SYSTEM test
  (* Version 1.0, 2022-11-09, franz *)
  APPLICATION testApp
  END_APPLICATION
  APPLICATION mapping_DataPanel
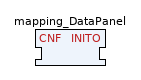
    SUBAPPLICATION mapping_DataPanel (* mapping_DataPanel *)
      EVENT_INPUT
        CNF;
      END_EVENT
      EVENT_OUTPUT
        INITO;
      END_EVENT
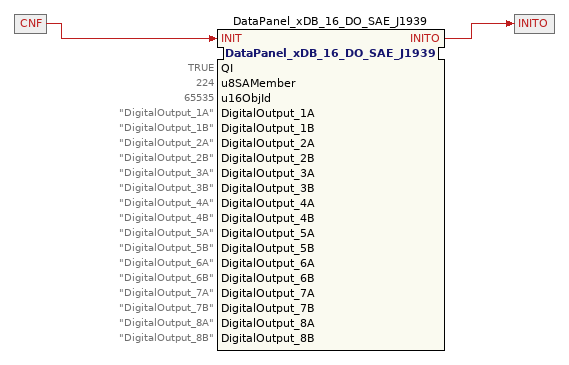
      FBS
        DataPanel_xDB_16_DO_SAE_J1939 : DataPanel_xDB_16_DO_SAE_J1939(QI := TRUE, u8SAMember := 224, u16ObjId := 65535, DigitalOutput_1A := "DigitalOutput_1A", DigitalOutput_1B := "DigitalOutput_1B", DigitalOutput_2A := "DigitalOutput_2A", DigitalOutput_2B := "DigitalOutput_2B", DigitalOutput_3A := "DigitalOutput_3A", DigitalOutput_3B := "DigitalOutput_3B", DigitalOutput_4A := "DigitalOutput_4A", DigitalOutput_4B := "DigitalOutput_4B", DigitalOutput_5A := "DigitalOutput_5A", DigitalOutput_5B := "DigitalOutput_5B", DigitalOutput_6A := "DigitalOutput_6A", DigitalOutput_6B := "DigitalOutput_6B", DigitalOutput_7A := "DigitalOutput_7A", DigitalOutput_7B := "DigitalOutput_7B", DigitalOutput_8A := "DigitalOutput_8A", DigitalOutput_8B := "DigitalOutput_8B");
      END_FBS
      EVENT_CONNECTIONS
        CNF TO DataPanel_xDB_16_DO_SAE_J1939.INIT;
        DataPanel_xDB_16_DO_SAE_J1939.INITO TO INITO;
      END_CONNECTIONS
    END_SUBAPPLICATION
  END_APPLICATION
  APPLICATION mapping_Softkeys
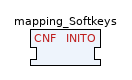
    SUBAPPLICATION mapping_Softkeys (* mapping_Softkeys *)
      EVENT_INPUT
        CNF;
      END_EVENT
      EVENT_OUTPUT
        INITO;
      END_EVENT
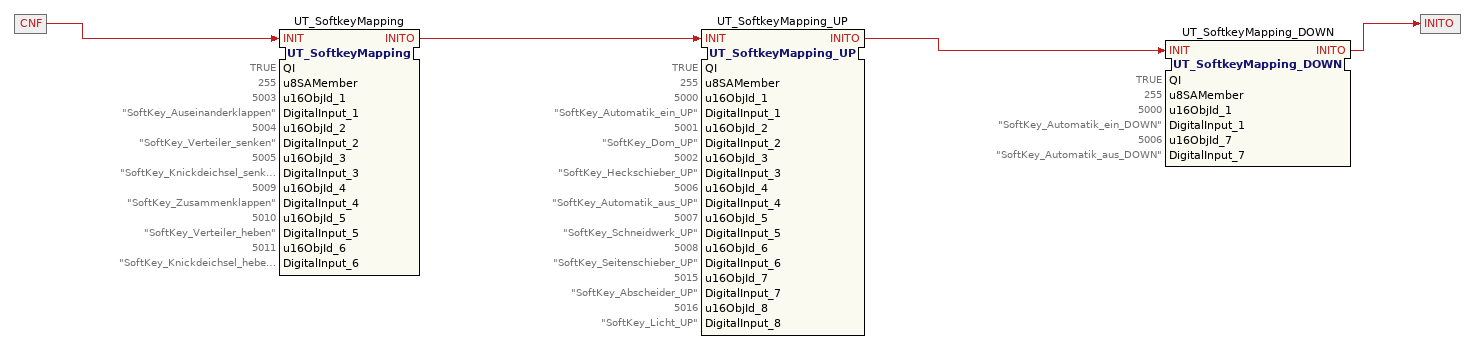
      FBS
        UT_SoftkeyMapping_DOWN : UT_SoftkeyMapping_DOWN(QI := TRUE, u8SAMember := 255, u16ObjId_1 := 5000, DigitalInput_1 := "SoftKey_Automatik_ein_DOWN", u16ObjId_7 := 5006, DigitalInput_7 := "SoftKey_Automatik_aus_DOWN");
        UT_SoftkeyMapping_UP : UT_SoftkeyMapping_UP(QI := TRUE, u8SAMember := 255, u16ObjId_1 := 5000, DigitalInput_1 := "SoftKey_Automatik_ein_UP", u16ObjId_2 := 5001, DigitalInput_2 := "SoftKey_Dom_UP", u16ObjId_3 := 5002, DigitalInput_3 := "SoftKey_Heckschieber_UP", u16ObjId_4 := 5006, DigitalInput_4 := "SoftKey_Automatik_aus_UP", u16ObjId_5 := 5007, DigitalInput_5 := "SoftKey_Schneidwerk_UP", u16ObjId_6 := 5008, DigitalInput_6 := "SoftKey_Seitenschieber_UP", u16ObjId_7 := 5015, DigitalInput_7 := "SoftKey_Abscheider_UP", u16ObjId_8 := 5016, DigitalInput_8 := "SoftKey_Licht_UP");
        UT_SoftkeyMapping : UT_SoftkeyMapping(QI := TRUE, u8SAMember := 255, u16ObjId_1 := 5003, DigitalInput_1 := "SoftKey_Auseinanderklappen", u16ObjId_2 := 5004, DigitalInput_2 := "SoftKey_Verteiler_senken", u16ObjId_3 := 5005, DigitalInput_3 := "SoftKey_Knickdeichsel_senken", u16ObjId_4 := 5009, DigitalInput_4 := "SoftKey_Zusammenklappen", u16ObjId_5 := 5010, DigitalInput_5 := "SoftKey_Verteiler_heben", u16ObjId_6 := 5011, DigitalInput_6 := "SoftKey_Knickdeichsel_heben");
      END_FBS
      EVENT_CONNECTIONS
        UT_SoftkeyMapping_UP.INITO TO UT_SoftkeyMapping_DOWN.INIT;
        UT_SoftkeyMapping.INITO TO UT_SoftkeyMapping_UP.INIT;
        UT_SoftkeyMapping_DOWN.INITO TO INITO;
        CNF TO UT_SoftkeyMapping.INIT;
      END_CONNECTIONS
    END_SUBAPPLICATION
  END_APPLICATION
  APPLICATION Klappen
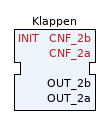
    SUBAPPLICATION Klappen (* Klappen *)
      EVENT_INPUT
        INIT;
      END_EVENT
      EVENT_OUTPUT
        CNF_2b;
        CNF_2a;
      END_EVENT
      VAR_OUTPUT
        OUT_2b : BOOL;
        OUT_2a : BOOL;
      END_VAR
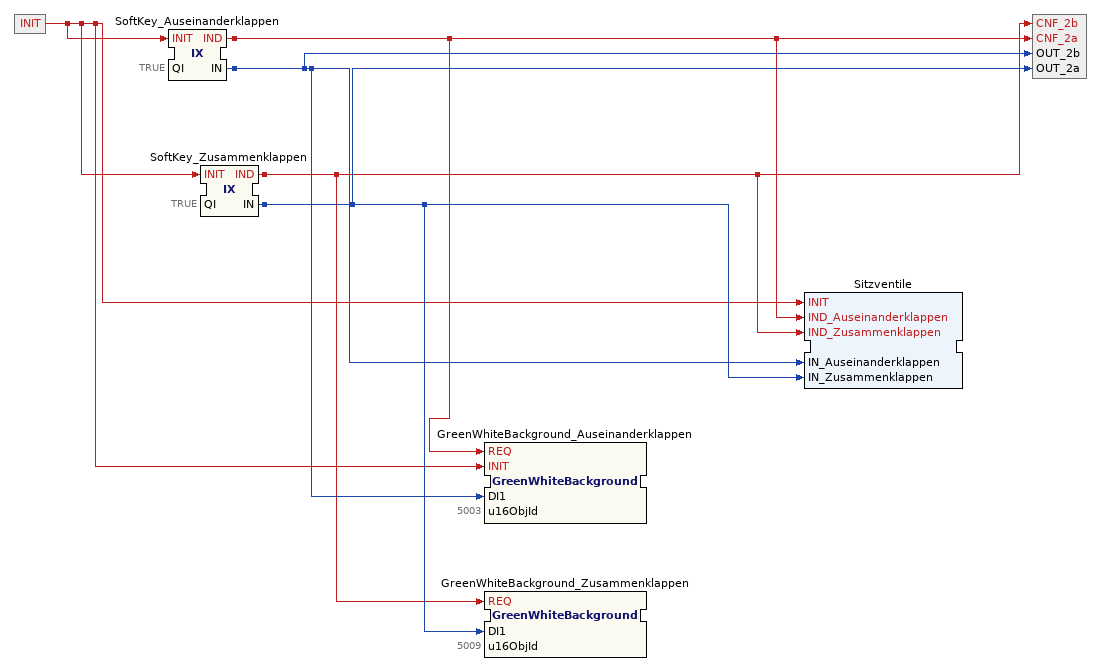
      FBS
        SoftKey_Auseinanderklappen : IX(QI := TRUE);
        GreenWhiteBackground_Auseinanderklappen : GreenWhiteBackground(u16ObjId := 5003);
        SoftKey_Zusammenklappen : IX(QI := TRUE);
        GreenWhiteBackground_Zusammenklappen : GreenWhiteBackground(u16ObjId := 5009);
      END_FBS
      SUBAPPLICATION Sitzventile (* Sitzventile *)
        EVENT_INPUT
          INIT;
          IND_Auseinanderklappen;
          IND_Zusammenklappen;
        END_EVENT
        VAR_INPUT
          IN_Auseinanderklappen : BOOL;
          IN_Zusammenklappen : BOOL;
        END_VAR
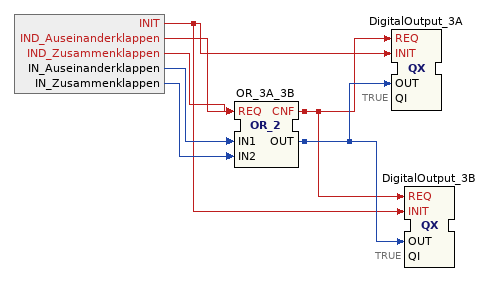
        FBS
          DigitalOutput_3B : QX(QI := TRUE);
          DigitalOutput_3A : QX(QI := TRUE);
          OR_3A_3B : OR_2; {SET_ATTRIBUTE(PinComment, IN1:Auseinanderklappen)} {SET_ATTRIBUTE(PinComment, IN2:Zusammenklappen)}
        END_FBS
        EVENT_CONNECTIONS
          OR_3A_3B.CNF TO DigitalOutput_3B.REQ;
          OR_3A_3B.CNF TO DigitalOutput_3A.REQ;
          INIT TO DigitalOutput_3B.INIT;
          INIT TO DigitalOutput_3A.INIT;
          IND_Auseinanderklappen TO OR_3A_3B.REQ;
          IND_Zusammenklappen TO OR_3A_3B.REQ;
        END_CONNECTIONS
        DATA_CONNECTIONS
          OR_3A_3B.OUT TO DigitalOutput_3B.OUT;
          OR_3A_3B.OUT TO DigitalOutput_3A.OUT;
          IN_Auseinanderklappen TO OR_3A_3B.IN1;
          IN_Zusammenklappen TO OR_3A_3B.IN2;
        END_CONNECTIONS
      END_SUBAPPLICATION
      EVENT_CONNECTIONS
        SoftKey_Auseinanderklappen.IND TO GreenWhiteBackground_Auseinanderklappen.REQ;
        INIT TO SoftKey_Auseinanderklappen.INIT;
        SoftKey_Auseinanderklappen.IND TO CNF_2b;
        INIT TO SoftKey_Zusammenklappen.INIT;
        SoftKey_Zusammenklappen.IND TO CNF_2a;
        INIT TO GreenWhiteBackground_Auseinanderklappen.INIT;
        INIT TO Sitzventile.INIT;
        SoftKey_Auseinanderklappen.IND TO Sitzventile.IND_Auseinanderklappen;
        SoftKey_Zusammenklappen.IND TO Sitzventile.IND_Zusammenklappen;
        SoftKey_Zusammenklappen.IND TO GreenWhiteBackground_Zusammenklappen.REQ;
      END_CONNECTIONS
      DATA_CONNECTIONS
        SoftKey_Auseinanderklappen.IN TO GreenWhiteBackground_Auseinanderklappen.DI1;
        SoftKey_Auseinanderklappen.IN TO OUT_2b;
        SoftKey_Zusammenklappen.IN TO OUT_2a;
        SoftKey_Auseinanderklappen.IN TO Sitzventile.IN_Auseinanderklappen;
        SoftKey_Zusammenklappen.IN TO Sitzventile.IN_Zusammenklappen;
        SoftKey_Zusammenklappen.IN TO GreenWhiteBackground_Zusammenklappen.DI1;
      END_CONNECTIONS
    END_SUBAPPLICATION
  END_APPLICATION
  APPLICATION Vorsteuerventil_2A
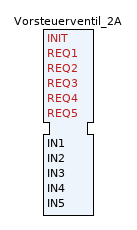
    SUBAPPLICATION Vorsteuerventil_2A (* Vorsteuerventil_2A *)
      EVENT_INPUT
        INIT;
        REQ1;
        REQ2;
        REQ3;
        REQ4;
        REQ5;
      END_EVENT
      VAR_INPUT
        IN1 : BOOL;
        IN2 : BOOL;
        IN3 : BOOL;
        IN4 : BOOL;
        IN5 : BOOL;
      END_VAR
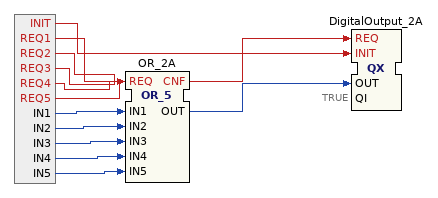
      FBS
        DigitalOutput_2A : QX(QI := TRUE);
        OR_2A : OR_5;
      END_FBS
      EVENT_CONNECTIONS
        OR_2A.CNF TO DigitalOutput_2A.REQ;
        INIT TO DigitalOutput_2A.INIT;
        REQ1 TO OR_2A.REQ;
        REQ2 TO OR_2A.REQ;
        REQ3 TO OR_2A.REQ;
        REQ4 TO OR_2A.REQ;
        REQ5 TO OR_2A.REQ;
      END_CONNECTIONS
      DATA_CONNECTIONS
        OR_2A.OUT TO DigitalOutput_2A.OUT;
        IN1 TO OR_2A.IN1;
        IN2 TO OR_2A.IN2;
        IN3 TO OR_2A.IN3;
        IN4 TO OR_2A.IN4;
        IN5 TO OR_2A.IN5;
      END_CONNECTIONS
    END_SUBAPPLICATION
  END_APPLICATION
  APPLICATION Verteiler
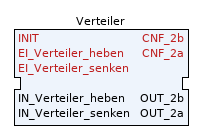
    SUBAPPLICATION Verteiler (* Verteiler *)
      EVENT_INPUT
        INIT;
        EI_Verteiler_heben;
        EI_Verteiler_senken;
      END_EVENT
      EVENT_OUTPUT
        CNF_2b;
        CNF_2a;
      END_EVENT
      VAR_INPUT
        IN_Verteiler_heben : BOOL;
        IN_Verteiler_senken : BOOL;
      END_VAR
      VAR_OUTPUT
        OUT_2b : BOOL;
        OUT_2a : BOOL;
      END_VAR
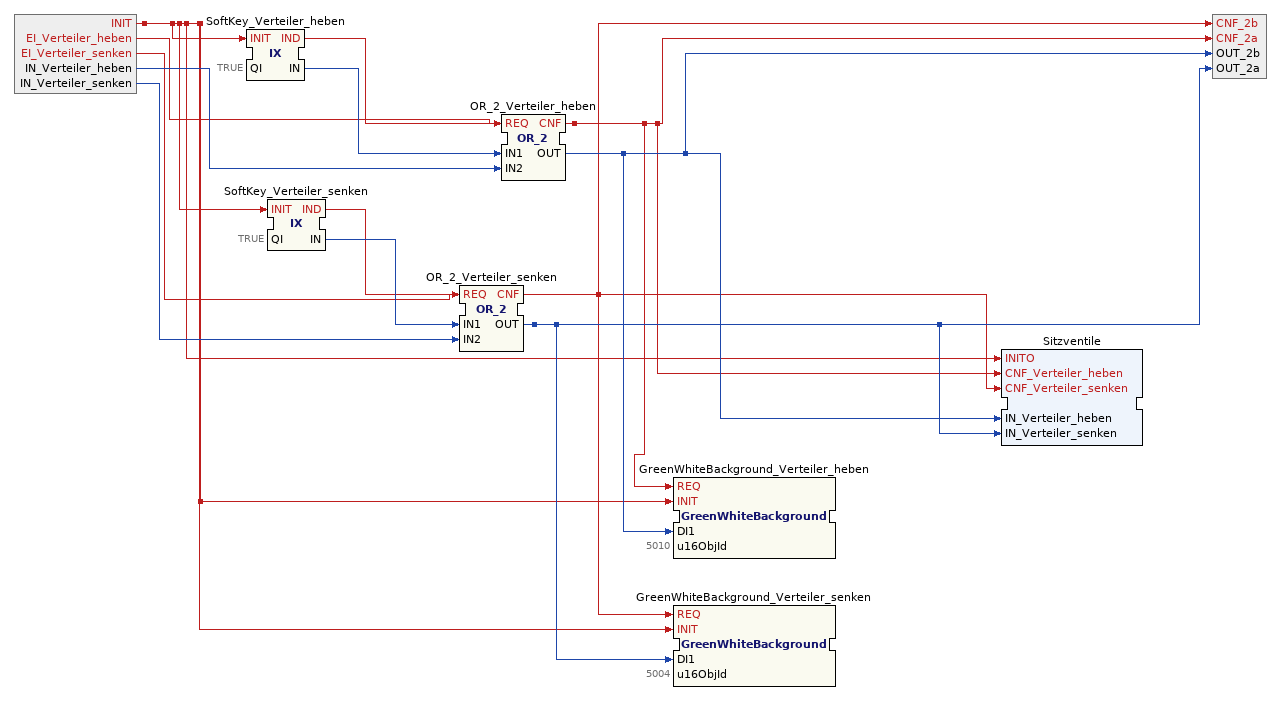
      FBS
        OR_2_Verteiler_senken : OR_2;
        SoftKey_Verteiler_heben : IX(QI := TRUE);
        OR_2_Verteiler_heben : OR_2;
        GreenWhiteBackground_Verteiler_heben : GreenWhiteBackground(u16ObjId := 5010);
        SoftKey_Verteiler_senken : IX(QI := TRUE);
        GreenWhiteBackground_Verteiler_senken : GreenWhiteBackground(u16ObjId := 5004);
      END_FBS
      SUBAPPLICATION Sitzventile (* Sitzventile *)
        EVENT_INPUT
          INITO;
          CNF_Verteiler_heben;
          CNF_Verteiler_senken;
        END_EVENT
        VAR_INPUT
          IN_Verteiler_heben : BOOL;
          IN_Verteiler_senken : BOOL;
        END_VAR
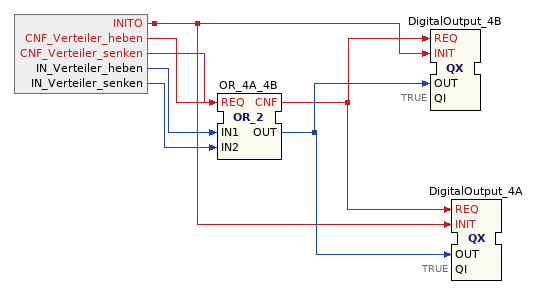
        FBS
          OR_4A_4B : OR_2; {SET_ATTRIBUTE(PinComment, IN1:Verteiler_heben)} {SET_ATTRIBUTE(PinComment, IN2:Verteiler_senken)}
          DigitalOutput_4B : QX(QI := TRUE);
          DigitalOutput_4A : QX(QI := TRUE);
        END_FBS
        EVENT_CONNECTIONS
          OR_4A_4B.CNF TO DigitalOutput_4B.REQ;
          OR_4A_4B.CNF TO DigitalOutput_4A.REQ;
          CNF_Verteiler_heben TO OR_4A_4B.REQ;
          CNF_Verteiler_senken TO OR_4A_4B.REQ;
          INITO TO DigitalOutput_4B.INIT;
          INITO TO DigitalOutput_4A.INIT;
        END_CONNECTIONS
        DATA_CONNECTIONS
          OR_4A_4B.OUT TO DigitalOutput_4B.OUT;
          OR_4A_4B.OUT TO DigitalOutput_4A.OUT;
          IN_Verteiler_heben TO OR_4A_4B.IN1;
          IN_Verteiler_senken TO OR_4A_4B.IN2;
        END_CONNECTIONS
      END_SUBAPPLICATION
      EVENT_CONNECTIONS
        SoftKey_Verteiler_senken.IND TO OR_2_Verteiler_senken.REQ;
        SoftKey_Verteiler_heben.IND TO OR_2_Verteiler_heben.REQ;
        OR_2_Verteiler_heben.CNF TO GreenWhiteBackground_Verteiler_heben.REQ;
        INIT TO SoftKey_Verteiler_heben.INIT;
        INIT TO SoftKey_Verteiler_senken.INIT;
        INIT TO Sitzventile.INITO;
        OR_2_Verteiler_senken.CNF TO GreenWhiteBackground_Verteiler_senken.REQ;
        INIT TO GreenWhiteBackground_Verteiler_heben.INIT;
        INIT TO GreenWhiteBackground_Verteiler_senken.INIT;
        OR_2_Verteiler_heben.CNF TO CNF_2a;
        OR_2_Verteiler_senken.CNF TO CNF_2b;
        OR_2_Verteiler_heben.CNF TO Sitzventile.CNF_Verteiler_heben;
        OR_2_Verteiler_senken.CNF TO Sitzventile.CNF_Verteiler_senken;
        EI_Verteiler_heben TO OR_2_Verteiler_heben.REQ;
        EI_Verteiler_senken TO OR_2_Verteiler_senken.REQ;
      END_CONNECTIONS
      DATA_CONNECTIONS
        SoftKey_Verteiler_senken.IN TO OR_2_Verteiler_senken.IN1;
        SoftKey_Verteiler_heben.IN TO OR_2_Verteiler_heben.IN1;
        OR_2_Verteiler_heben.OUT TO GreenWhiteBackground_Verteiler_heben.DI1;
        IN_Verteiler_senken TO OR_2_Verteiler_senken.IN2;
        IN_Verteiler_heben TO OR_2_Verteiler_heben.IN2;
        OR_2_Verteiler_heben.OUT TO Sitzventile.IN_Verteiler_heben;
        OR_2_Verteiler_senken.OUT TO Sitzventile.IN_Verteiler_senken;
        OR_2_Verteiler_senken.OUT TO GreenWhiteBackground_Verteiler_senken.DI1;
        OR_2_Verteiler_heben.OUT TO OUT_2b;
        OR_2_Verteiler_senken.OUT TO OUT_2a;
      END_CONNECTIONS
    END_SUBAPPLICATION
  END_APPLICATION
  APPLICATION Knickdeichsel
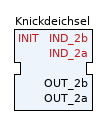
    SUBAPPLICATION Knickdeichsel (* Knickdeichsel *)
      EVENT_INPUT
        INIT;
      END_EVENT
      EVENT_OUTPUT
        IND_2b;
        IND_2a;
      END_EVENT
      VAR_OUTPUT
        OUT_2b : BOOL;
        OUT_2a : BOOL;
      END_VAR
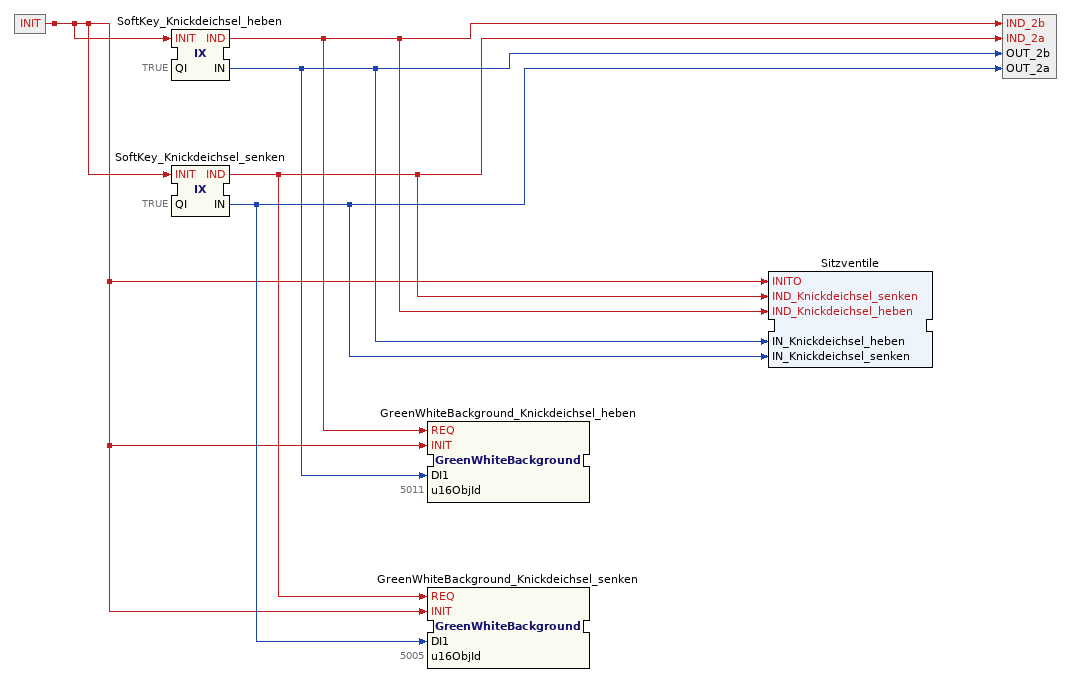
      FBS
        SoftKey_Knickdeichsel_heben : IX(QI := TRUE);
        SoftKey_Knickdeichsel_senken : IX(QI := TRUE);
        GreenWhiteBackground_Knickdeichsel_senken : GreenWhiteBackground(u16ObjId := 5005);
        GreenWhiteBackground_Knickdeichsel_heben : GreenWhiteBackground(u16ObjId := 5011);
      END_FBS
      SUBAPPLICATION Sitzventile (* Sitzventile *)
        EVENT_INPUT
          INITO;
          IND_Knickdeichsel_senken;
          IND_Knickdeichsel_heben;
        END_EVENT
        VAR_INPUT
          IN_Knickdeichsel_heben : BOOL;
          IN_Knickdeichsel_senken : BOOL;
        END_VAR
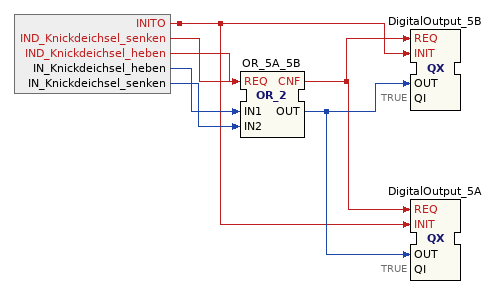
        FBS
          OR_5A_5B : OR_2; {SET_ATTRIBUTE(PinComment, IN1:Knickdeichsel_heben)} {SET_ATTRIBUTE(PinComment, IN2:Knickdeichsel_senken)}
          DigitalOutput_5B : QX(QI := TRUE);
          DigitalOutput_5A : QX(QI := TRUE);
        END_FBS
        EVENT_CONNECTIONS
          OR_5A_5B.CNF TO DigitalOutput_5B.REQ;
          OR_5A_5B.CNF TO DigitalOutput_5A.REQ;
          IND_Knickdeichsel_senken TO OR_5A_5B.REQ;
          IND_Knickdeichsel_heben TO OR_5A_5B.REQ;
          INITO TO DigitalOutput_5B.INIT;
          INITO TO DigitalOutput_5A.INIT;
        END_CONNECTIONS
        DATA_CONNECTIONS
          OR_5A_5B.OUT TO DigitalOutput_5B.OUT;
          OR_5A_5B.OUT TO DigitalOutput_5A.OUT;
          IN_Knickdeichsel_heben TO OR_5A_5B.IN1;
          IN_Knickdeichsel_senken TO OR_5A_5B.IN2;
        END_CONNECTIONS
      END_SUBAPPLICATION
      EVENT_CONNECTIONS
        SoftKey_Knickdeichsel_heben.IND TO GreenWhiteBackground_Knickdeichsel_heben.REQ;
        SoftKey_Knickdeichsel_senken.IND TO GreenWhiteBackground_Knickdeichsel_senken.REQ;
        INIT TO SoftKey_Knickdeichsel_heben.INIT;
        SoftKey_Knickdeichsel_heben.IND TO IND_2b;
        INIT TO SoftKey_Knickdeichsel_senken.INIT;
        SoftKey_Knickdeichsel_senken.IND TO IND_2a;
        SoftKey_Knickdeichsel_senken.IND TO Sitzventile.IND_Knickdeichsel_senken;
        SoftKey_Knickdeichsel_heben.IND TO Sitzventile.IND_Knickdeichsel_heben;
        INIT TO Sitzventile.INITO;
        INIT TO GreenWhiteBackground_Knickdeichsel_heben.INIT;
        INIT TO GreenWhiteBackground_Knickdeichsel_senken.INIT;
      END_CONNECTIONS
      DATA_CONNECTIONS
        SoftKey_Knickdeichsel_heben.IN TO GreenWhiteBackground_Knickdeichsel_heben.DI1;
        SoftKey_Knickdeichsel_senken.IN TO GreenWhiteBackground_Knickdeichsel_senken.DI1;
        SoftKey_Knickdeichsel_heben.IN TO OUT_2b;
        SoftKey_Knickdeichsel_senken.IN TO OUT_2a;
        SoftKey_Knickdeichsel_heben.IN TO Sitzventile.IN_Knickdeichsel_heben;
        SoftKey_Knickdeichsel_senken.IN TO Sitzventile.IN_Knickdeichsel_senken;
      END_CONNECTIONS
    END_SUBAPPLICATION
  END_APPLICATION
  APPLICATION Dom
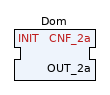
    SUBAPPLICATION Dom (* Dom *)
      EVENT_INPUT
        INIT;
      END_EVENT
      EVENT_OUTPUT
        CNF_2a;
      END_EVENT
      VAR_OUTPUT
        OUT_2a : BOOL;
      END_VAR
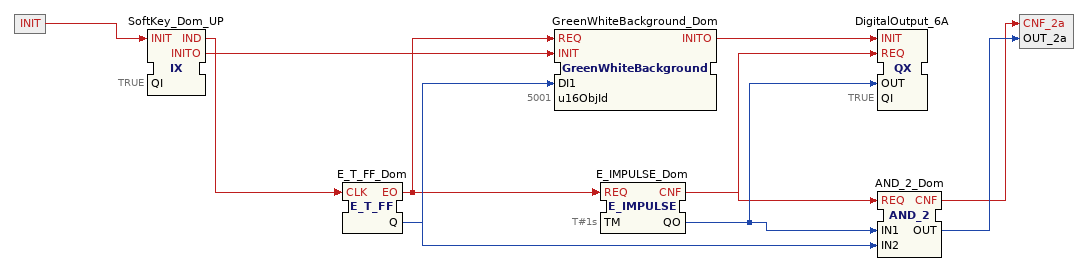
      FBS
        AND_2_Dom : AND_2;
        E_T_FF_Dom : E_T_FF;
        DigitalOutput_6A : QX(QI := TRUE);
        GreenWhiteBackground_Dom : GreenWhiteBackground(u16ObjId := 5001);
        E_IMPULSE_Dom : E_IMPULSE(TM := T#1s);
        SoftKey_Dom_UP : IX(QI := TRUE);
      END_FBS
      EVENT_CONNECTIONS
        E_IMPULSE_Dom.CNF TO AND_2_Dom.REQ;
        SoftKey_Dom_UP.IND TO E_T_FF_Dom.CLK;
        E_T_FF_Dom.EO TO GreenWhiteBackground_Dom.REQ;
        E_T_FF_Dom.EO TO E_IMPULSE_Dom.REQ;
        GreenWhiteBackground_Dom.INITO TO DigitalOutput_6A.INIT;
        E_IMPULSE_Dom.CNF TO DigitalOutput_6A.REQ;
        SoftKey_Dom_UP.INITO TO GreenWhiteBackground_Dom.INIT;
        AND_2_Dom.CNF TO CNF_2a;
        INIT TO SoftKey_Dom_UP.INIT;
      END_CONNECTIONS
      DATA_CONNECTIONS
        E_IMPULSE_Dom.QO TO AND_2_Dom.IN1;
        E_T_FF_Dom.Q TO AND_2_Dom.IN2;
        E_T_FF_Dom.Q TO GreenWhiteBackground_Dom.DI1;
        E_IMPULSE_Dom.QO TO DigitalOutput_6A.OUT;
        AND_2_Dom.OUT TO OUT_2a;
      END_CONNECTIONS
    END_SUBAPPLICATION
  END_APPLICATION
  APPLICATION Heckschieber
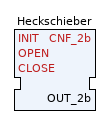
    SUBAPPLICATION Heckschieber (* Heckschieber *)
      EVENT_INPUT
        INIT;
        OPEN;
        CLOSE;
      END_EVENT
      EVENT_OUTPUT
        CNF_2b;
      END_EVENT
      VAR_OUTPUT
        OUT_2b : BOOL;
      END_VAR
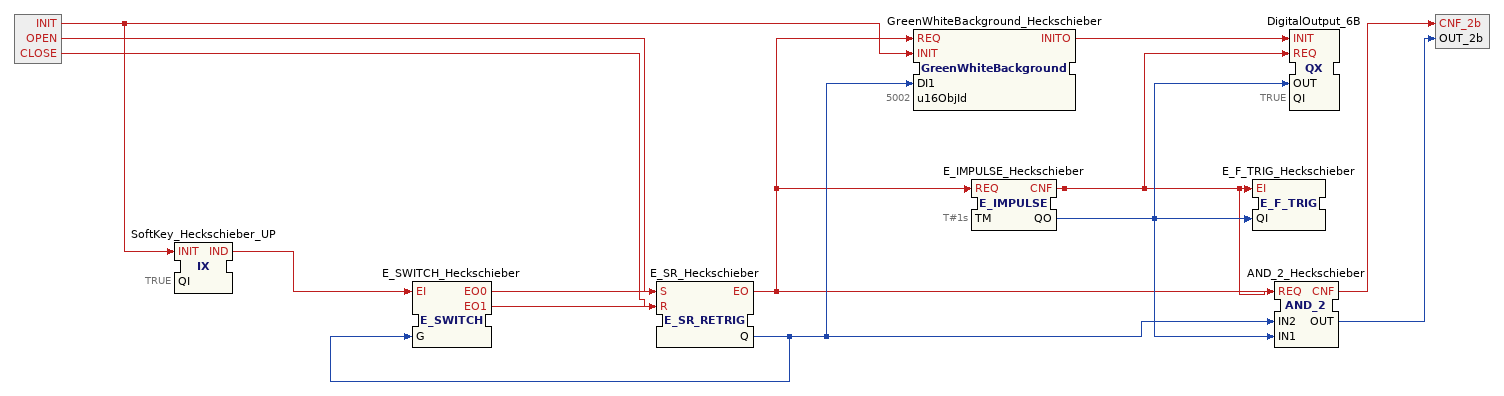
      FBS
        E_F_TRIG_Heckschieber : E_F_TRIG;
        GreenWhiteBackground_Heckschieber : GreenWhiteBackground(u16ObjId := 5002);
        SoftKey_Heckschieber_UP : IX(QI := TRUE);
        DigitalOutput_6B : QX(QI := TRUE);
        E_SR_Heckschieber : E_SR_RETRIG;
        E_SWITCH_Heckschieber : E_SWITCH;
        AND_2_Heckschieber : AND_2;
        E_IMPULSE_Heckschieber : E_IMPULSE(TM := T#1s);
      END_FBS
      EVENT_CONNECTIONS
        E_IMPULSE_Heckschieber.CNF TO E_F_TRIG_Heckschieber.EI;
        E_SR_Heckschieber.EO TO GreenWhiteBackground_Heckschieber.REQ;
        GreenWhiteBackground_Heckschieber.INITO TO DigitalOutput_6B.INIT;
        SoftKey_Heckschieber_UP.IND TO E_SWITCH_Heckschieber.EI;
        E_IMPULSE_Heckschieber.CNF TO DigitalOutput_6B.REQ;
        E_SWITCH_Heckschieber.EO0 TO E_SR_Heckschieber.S;
        E_SWITCH_Heckschieber.EO1 TO E_SR_Heckschieber.R;
        E_SR_Heckschieber.EO TO AND_2_Heckschieber.REQ;
        E_SR_Heckschieber.EO TO E_IMPULSE_Heckschieber.REQ;
        E_IMPULSE_Heckschieber.CNF TO AND_2_Heckschieber.REQ;
        INIT TO SoftKey_Heckschieber_UP.INIT;
        OPEN TO E_SR_Heckschieber.S;
        CLOSE TO E_SR_Heckschieber.R;
        AND_2_Heckschieber.CNF TO CNF_2b;
        INIT TO GreenWhiteBackground_Heckschieber.INIT;
      END_CONNECTIONS
      DATA_CONNECTIONS
        E_IMPULSE_Heckschieber.QO TO E_F_TRIG_Heckschieber.QI;
        E_SR_Heckschieber.Q TO GreenWhiteBackground_Heckschieber.DI1;
        E_IMPULSE_Heckschieber.QO TO DigitalOutput_6B.OUT;
        E_SR_Heckschieber.Q TO E_SWITCH_Heckschieber.G;
        E_SR_Heckschieber.Q TO AND_2_Heckschieber.IN2;
        E_IMPULSE_Heckschieber.QO TO AND_2_Heckschieber.IN1;
        AND_2_Heckschieber.OUT TO OUT_2b;
      END_CONNECTIONS
    END_SUBAPPLICATION
  END_APPLICATION
  APPLICATION Seitenschieber
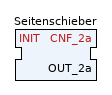
    SUBAPPLICATION Seitenschieber (* Seitenschieber *)
      EVENT_INPUT
        INIT;
      END_EVENT
      EVENT_OUTPUT
        CNF_2a;
      END_EVENT
      VAR_OUTPUT
        OUT_2a : BOOL;
      END_VAR
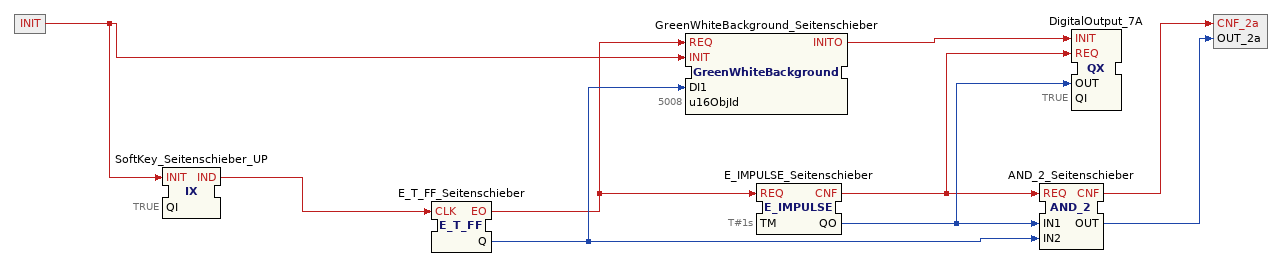
      FBS
        GreenWhiteBackground_Seitenschieber : GreenWhiteBackground(u16ObjId := 5008);
        E_IMPULSE_Seitenschieber : E_IMPULSE(TM := T#1s);
        AND_2_Seitenschieber : AND_2;
        E_T_FF_Seitenschieber : E_T_FF;
        SoftKey_Seitenschieber_UP : IX(QI := TRUE);
        DigitalOutput_7A : QX(QI := TRUE);
      END_FBS
      EVENT_CONNECTIONS
        E_T_FF_Seitenschieber.EO TO GreenWhiteBackground_Seitenschieber.REQ;
        GreenWhiteBackground_Seitenschieber.INITO TO DigitalOutput_7A.INIT;
        E_T_FF_Seitenschieber.EO TO E_IMPULSE_Seitenschieber.REQ;
        E_IMPULSE_Seitenschieber.CNF TO DigitalOutput_7A.REQ;
        E_IMPULSE_Seitenschieber.CNF TO AND_2_Seitenschieber.REQ;
        SoftKey_Seitenschieber_UP.IND TO E_T_FF_Seitenschieber.CLK;
        AND_2_Seitenschieber.CNF TO CNF_2a;
        INIT TO SoftKey_Seitenschieber_UP.INIT;
        INIT TO GreenWhiteBackground_Seitenschieber.INIT;
      END_CONNECTIONS
      DATA_CONNECTIONS
        E_T_FF_Seitenschieber.Q TO GreenWhiteBackground_Seitenschieber.DI1;
        E_IMPULSE_Seitenschieber.QO TO AND_2_Seitenschieber.IN1;
        E_IMPULSE_Seitenschieber.QO TO DigitalOutput_7A.OUT;
        E_T_FF_Seitenschieber.Q TO AND_2_Seitenschieber.IN2;
        AND_2_Seitenschieber.OUT TO OUT_2a;
      END_CONNECTIONS
    END_SUBAPPLICATION
  END_APPLICATION
  APPLICATION Schneidwerk
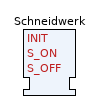
    SUBAPPLICATION Schneidwerk (* Schneidwerk *)
      EVENT_INPUT
        INIT;
        S_ON;
        S_OFF;
      END_EVENT
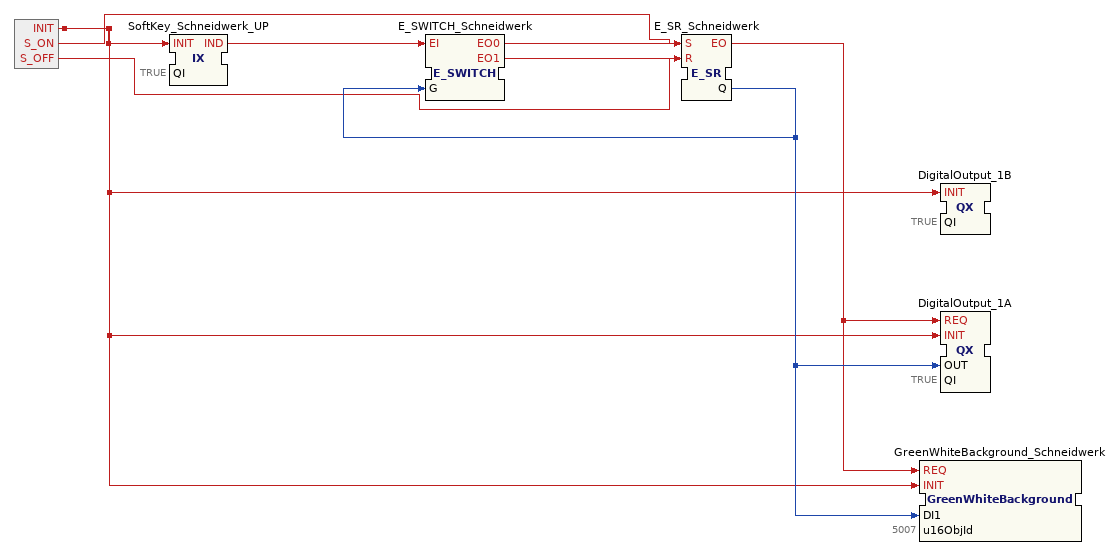
      FBS
        DigitalOutput_1A : QX(QI := TRUE);
        GreenWhiteBackground_Schneidwerk : GreenWhiteBackground(u16ObjId := 5007);
        SoftKey_Schneidwerk_UP : IX(QI := TRUE);
        E_SWITCH_Schneidwerk : E_SWITCH;
        E_SR_Schneidwerk : E_SR;
        DigitalOutput_1B : QX(QI := TRUE);
      END_FBS
      EVENT_CONNECTIONS
        E_SR_Schneidwerk.EO TO DigitalOutput_1A.REQ;
        E_SR_Schneidwerk.EO TO GreenWhiteBackground_Schneidwerk.REQ;
        SoftKey_Schneidwerk_UP.IND TO E_SWITCH_Schneidwerk.EI;
        E_SWITCH_Schneidwerk.EO0 TO E_SR_Schneidwerk.S;
        E_SWITCH_Schneidwerk.EO1 TO E_SR_Schneidwerk.R;
        INIT TO SoftKey_Schneidwerk_UP.INIT;
        S_ON TO E_SR_Schneidwerk.S;
        S_OFF TO E_SR_Schneidwerk.R;
        INIT TO DigitalOutput_1B.INIT;
        INIT TO GreenWhiteBackground_Schneidwerk.INIT;
        INIT TO DigitalOutput_1A.INIT;
      END_CONNECTIONS
      DATA_CONNECTIONS
        E_SR_Schneidwerk.Q TO DigitalOutput_1A.OUT;
        E_SR_Schneidwerk.Q TO GreenWhiteBackground_Schneidwerk.DI1;
        E_SR_Schneidwerk.Q TO E_SWITCH_Schneidwerk.G;
      END_CONNECTIONS
    END_SUBAPPLICATION
  END_APPLICATION
  APPLICATION Licht
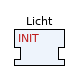
    SUBAPPLICATION Licht (* Licht *)
      EVENT_INPUT
        INIT; (* Service Initialization *)
      END_EVENT
